(* PLC project prj, KAIST_DSLAB noNameNow 1, author bwkim *)
(* stored: creationDateTime 2018-0-3T10:17:27, modificationDateTime 2018-0-3T10:17:30 *)

PROGRAM program7____wholeTest
  VAR
    FR_PTRIP_TON_copy : null;
  END_VAR
  VAR
    FR_TRIP_TON_copy : null;
  END_VAR
  VAR
    PTRIP_TON : null;
  END_VAR
  VAR
    TRIP_TON : null;
  END_VAR
  VAR
    PTRIP_TON_copy : null;
  END_VAR
  VAR
    TRIP_TON_copy : null;
  END_VAR
  VAR
    PTRIP_TON_copy_copy : null;
  END_VAR
  VAR
    TRIP_TON_copy_copy : null;
  END_VAR
  VAR
    FR_PTRIP_TON_copy_copy : null;
  END_VAR
  VAR
    FR_TRIP_TON_copy_copy : null;
  END_VAR
  VAR
    VF_PTON_copy : null;
  END_VAR
  VAR
    VF_TON_copy : null;
  END_VAR
  VAR
    FR_PTRIP_TON_copy_copy_copy : null;
  END_VAR
  VAR
    FR_TRIP_TON_copy_copy_copy : null;
  END_VAR
  VAR
    FR_PTRIP_TON_copy_copy_copy_copy : null;
  END_VAR
  VAR
    FR_TRIP_TON_copy_copy_copy_copy : null;
  END_VAR
  VAR
    VF_PTON_copy_copy : null;
  END_VAR
  VAR
    VF_TON_copy_copy : null;
  END_VAR
  VAR
    PTRIP_TON_copy_copy_copy : null;
  END_VAR
  VAR
    TRIP_TON_copy_copy_copy : null;
  END_VAR
  VAR
    PTRIP_TON_copy_copy_copy_copy : null;
  END_VAR
  VAR
    TRIP_TON_copy_copy_copy_copy : null;
  END_VAR
  VAR
    FR_PTRIP_TON_copy_copy_copy_copy_copy : null;
  END_VAR
  VAR
    FR_TRIP_TON_copy_copy_copy_copy_copy : null;
  END_VAR
  VAR
    VF_PTON_copy_copy_copy : null;
  END_VAR
  VAR
    VF_TON_copy_copy_copy : null;
  END_VAR
  VAR
    FR_PTRIP_TON_copy_copy_copy_copy_copy_copy : null;
  END_VAR
  VAR
    FR_TRIP_TON_copy_copy_copy_copy_copy_copy : null;
  END_VAR
  VAR_INPUT
    _5_PV_OUT : BOOL := FALSE;
  END_VAR
  VAR_INPUT
    _5_K_DELAY : BOOL := FALSE;
  END_VAR
  VAR_INPUT
    _5_PHYS : BOOL := FALSE;
  END_VAR
  VAR_INPUT
    _5_HYS : BOOL := FALSE;
  END_VAR
  VAR_INPUT
    _5_RNG_MIN : BOOL := FALSE;
  END_VAR
  VAR_INPUT
    _5_RNG_MAX : BOOL := FALSE;
  END_VAR
  VAR_INPUT
    _5_MDL_E : BOOL := FALSE;
  END_VAR
  VAR_INPUT
    _5_AI_E : BOOL := FALSE;
  END_VAR
  VAR_INPUT
    _5_OB_INIT_STA : BOOL := FALSE;
  END_VAR
  VAR_INPUT
    _7_PV_OUT : BOOL := FALSE;
  END_VAR
  VAR_INPUT
    _7_PHYS : BOOL := FALSE;
  END_VAR
  VAR_INPUT
    _7_K_DELAY : BOOL := FALSE;
  END_VAR
  VAR_INPUT
    _7_HYS : BOOL := FALSE;
  END_VAR
  VAR_INPUT
    _7_RNG_MIN : BOOL := FALSE;
  END_VAR
  VAR_INPUT
    _7_RNG_MAX : BOOL := FALSE;
  END_VAR
  VAR_INPUT
    _7_MDL_E : BOOL := FALSE;
  END_VAR
  VAR_INPUT
    _7_AI_E : BOOL := FALSE;
  END_VAR
  VAR_INPUT
    _7_OB_INIT_STA : BOOL := FALSE;
  END_VAR
  VAR_INPUT
    _9_PV_OUT : BOOL := FALSE;
  END_VAR
  VAR_INPUT
    _9_PK_DELAY : BOOL := FALSE;
  END_VAR
  VAR_INPUT
    _9_PHYS : BOOL := FALSE;
  END_VAR
  VAR_INPUT
    _9_K_DELAY : BOOL := FALSE;
  END_VAR
  VAR_INPUT
    _9_HYS : BOOL := FALSE;
  END_VAR
  VAR_INPUT
    _9_RNG_MIN : BOOL := FALSE;
  END_VAR
  VAR_INPUT
    _9_RNG_MAX : BOOL := FALSE;
  END_VAR
  VAR_INPUT
    _9_MDL_E : BOOL := FALSE;
  END_VAR
  VAR_INPUT
    _9_AI_E : BOOL := FALSE;
  END_VAR
  VAR_INPUT
    _9_OB_INIT_STA : BOOL := FALSE;
  END_VAR
  VAR_INPUT
    _B_PV_OUT : BOOL := FALSE;
  END_VAR
  VAR_INPUT
    _B_K_DELAY : BOOL := FALSE;
  END_VAR
  VAR_INPUT
    _B_HYS : BOOL := FALSE;
  END_VAR
  VAR_INPUT
    _B_RNG_MIN : BOOL := FALSE;
  END_VAR
  VAR_INPUT
    _B_RNG_MAX : BOOL := FALSE;
  END_VAR
  VAR_INPUT
    _B_MDL_E : BOOL := FALSE;
  END_VAR
  VAR_INPUT
    _B_AI_E : BOOL := FALSE;
  END_VAR
  VAR_INPUT
    _B_OB_INIT_STA : BOOL := FALSE;
  END_VAR
  VAR_INPUT
    _D_RATE_LMT : BOOL := FALSE;
  END_VAR
  VAR_INPUT
    _D_PV_OUT : BOOL := FALSE;
  END_VAR
  VAR_INPUT
    _D_PV2TSP_DIFF : BOOL := FALSE;
  END_VAR
  VAR_INPUT
    _D_TSP_PRETRIP : BOOL := FALSE;
  END_VAR
  VAR_INPUT
    _D_RATE_TSP_MIN : BOOL := FALSE;
  END_VAR
  VAR_INPUT
    _D_PTSP_PRETRIP : BOOL := FALSE;
  END_VAR
  VAR_INPUT
    _D_TSP2PTSP_DIFF : BOOL := FALSE;
  END_VAR
  VAR_INPUT
    _D_HYS : BOOL := FALSE;
  END_VAR
  VAR_INPUT
    _D_RNG_MIN : BOOL := FALSE;
  END_VAR
  VAR_INPUT
    _D_RNG_MAX : BOOL := FALSE;
  END_VAR
  VAR_INPUT
    _D_MDL_E : BOOL := FALSE;
  END_VAR
  VAR_INPUT
    _D_AI_E : BOOL := FALSE;
  END_VAR
  VAR_INPUT
    _D_OB_INIT_STA : BOOL := FALSE;
  END_VAR
  VAR_INPUT
    _F_PV_OUT : BOOL := FALSE;
  END_VAR
  VAR_INPUT
    _F_K_DELAY : BOOL := FALSE;
  END_VAR
  VAR_INPUT
    _F_HYS : BOOL := FALSE;
  END_VAR
  VAR_INPUT
    _F_RNG_MIN : BOOL := FALSE;
  END_VAR
  VAR_INPUT
    _F_RNG_MAX : BOOL := FALSE;
  END_VAR
  VAR_INPUT
    _F_MDL_E : BOOL := FALSE;
  END_VAR
  VAR_INPUT
    _F_AI_E : BOOL := FALSE;
  END_VAR
  VAR_INPUT
    _F_OB_INIT_STA : BOOL := FALSE;
  END_VAR
  VAR_INPUT
    _G_PV_OUT : BOOL := FALSE;
  END_VAR
  VAR_INPUT
    _G_K_DELAY : BOOL := FALSE;
  END_VAR
  VAR_INPUT
    _G_PHYS : BOOL := FALSE;
  END_VAR
  VAR_INPUT
    _G_HYS : BOOL := FALSE;
  END_VAR
  VAR_INPUT
    _G_RNG_MIN : BOOL := FALSE;
  END_VAR
  VAR_INPUT
    _G_RNG_MAX : BOOL := FALSE;
  END_VAR
  VAR_INPUT
    _G_MDL_E : BOOL := FALSE;
  END_VAR
  VAR_INPUT
    _G_AI_E : BOOL := FALSE;
  END_VAR
  VAR_INPUT
    _G_OB_INIT_STA : BOOL := FALSE;
  END_VAR
  VAR_INPUT
    _6_RATE_LMT : BOOL := FALSE;
  END_VAR
  VAR_INPUT
    _6_PV_OUT : BOOL := FALSE;
  END_VAR
  VAR_INPUT
    _6_PV2TSP_DIFF : BOOL := FALSE;
  END_VAR
  VAR_INPUT
    _6_RATE_TSP_MIN : BOOL := FALSE;
  END_VAR
  VAR_INPUT
    _6_TSP2PTSP_DIFF : BOOL := FALSE;
  END_VAR
  VAR_INPUT
    _6_K_DELAY : BOOL := FALSE;
  END_VAR
  VAR_INPUT
    _6_HYS : BOOL := FALSE;
  END_VAR
  VAR_INPUT
    _6_RNG_MIN : BOOL := FALSE;
  END_VAR
  VAR_INPUT
    _6_RNG_MAX : BOOL := FALSE;
  END_VAR
  VAR_INPUT
    _6_MDL_E : BOOL := FALSE;
  END_VAR
  VAR_INPUT
    _6_AI_E : BOOL := FALSE;
  END_VAR
  VAR_INPUT
    _6_OB_INIT_STA : BOOL := FALSE;
  END_VAR
  VAR_INPUT
    _8_PV_OUT : BOOL := FALSE;
  END_VAR
  VAR_INPUT
    _8_PK_DELAY : BOOL := FALSE;
  END_VAR
  VAR_INPUT
    _8_PHYS : BOOL := FALSE;
  END_VAR
  VAR_INPUT
    _8_K_DELAY : BOOL := FALSE;
  END_VAR
  VAR_INPUT
    _8_HYS : BOOL := FALSE;
  END_VAR
  VAR_INPUT
    _8_RNG_MIN : BOOL := FALSE;
  END_VAR
  VAR_INPUT
    _8_RNG_MAX : BOOL := FALSE;
  END_VAR
  VAR_INPUT
    _8_MDL_E : BOOL := FALSE;
  END_VAR
  VAR_INPUT
    _8_AI_E : BOOL := FALSE;
  END_VAR
  VAR_INPUT
    _8_OB_INIT_STA : BOOL := FALSE;
  END_VAR
  VAR_INPUT
    _A_PV_OUT : BOOL := FALSE;
  END_VAR
  VAR_INPUT
    _A_PK_DELAY : BOOL := FALSE;
  END_VAR
  VAR_INPUT
    _A_PHYS : BOOL := FALSE;
  END_VAR
  VAR_INPUT
    _A_K_DELAY : BOOL := FALSE;
  END_VAR
  VAR_INPUT
    _A_HYS : BOOL := FALSE;
  END_VAR
  VAR_INPUT
    _A_RNG_MIN : BOOL := FALSE;
  END_VAR
  VAR_INPUT
    _A_RNG_MAX : BOOL := FALSE;
  END_VAR
  VAR_INPUT
    _A_MDL_E : BOOL := FALSE;
  END_VAR
  VAR_INPUT
    _A_AI_E : BOOL := FALSE;
  END_VAR
  VAR_INPUT
    _A_OB_INIT_STA : BOOL := FALSE;
  END_VAR
  VAR_INPUT
    _C_PV_OUT : BOOL := FALSE;
  END_VAR
  VAR_INPUT
    _C_K_DELAY : BOOL := FALSE;
  END_VAR
  VAR_INPUT
    _C_PHYS : BOOL := FALSE;
  END_VAR
  VAR_INPUT
    _C_HYS : BOOL := FALSE;
  END_VAR
  VAR_INPUT
    _C_RNG_MIN : BOOL := FALSE;
  END_VAR
  VAR_INPUT
    _C_RNG_MAX : BOOL := FALSE;
  END_VAR
  VAR_INPUT
    _C_MDL_E : BOOL := FALSE;
  END_VAR
  VAR_INPUT
    _C_AI_E : BOOL := FALSE;
  END_VAR
  VAR_INPUT
    _C_OB_INIT_STA : BOOL := FALSE;
  END_VAR
  VAR_INPUT
    _E_RATE_LMT : BOOL := FALSE;
  END_VAR
  VAR_INPUT
    _E_PV_OUT : BOOL := FALSE;
  END_VAR
  VAR_INPUT
    _E_PV2TSP_DIFF : BOOL := FALSE;
  END_VAR
  VAR_INPUT
    _E_TSP_PRETRIP : BOOL := FALSE;
  END_VAR
  VAR_INPUT
    _E_RATE_TSP_MIN : BOOL := FALSE;
  END_VAR
  VAR_INPUT
    _E_PTSP_PRETRIP : BOOL := FALSE;
  END_VAR
  VAR_INPUT
    _E_TSP2PTSP_DIFF : BOOL := FALSE;
  END_VAR
  VAR_INPUT
    _E_K_DELAY : BOOL := FALSE;
  END_VAR
  VAR_INPUT
    _E_HYS : BOOL := FALSE;
  END_VAR
  VAR_INPUT
    _E_RNG_MIN : BOOL := FALSE;
  END_VAR
  VAR_INPUT
    _E_RNG_MAX : BOOL := FALSE;
  END_VAR
  VAR_INPUT
    _E_MDL_E : BOOL := FALSE;
  END_VAR
  VAR_INPUT
    _E_AI_E : BOOL := FALSE;
  END_VAR
  VAR_INPUT
    _E_OB_INIT_STA : BOOL := FALSE;
  END_VAR
  VAR_INPUT
    _2_PV_OUT : BOOL := FALSE;
  END_VAR
  VAR_INPUT
    _2_K_DELAY : BOOL := FALSE;
  END_VAR
  VAR_INPUT
    _2_PHYS : BOOL := FALSE;
  END_VAR
  VAR_INPUT
    _2_HYS : BOOL := FALSE;
  END_VAR
  VAR_INPUT
    _2_RNG_MIN : BOOL := FALSE;
  END_VAR
  VAR_INPUT
    _2_RNG_MAX : BOOL := FALSE;
  END_VAR
  VAR_INPUT
    _2_MDL_E : BOOL := FALSE;
  END_VAR
  VAR_INPUT
    _2_AI_E : BOOL := FALSE;
  END_VAR
  VAR_INPUT
    _2_OB_INIT_STA : BOOL := FALSE;
  END_VAR
  VAR_OUTPUT
    _5_PTON_et : BOOL := FALSE;
  END_VAR
  VAR_OUTPUT
    _5_TON_et : BOOL := FALSE;
  END_VAR
  VAR_OUTPUT
    _7_TON_et : BOOL := FALSE;
  END_VAR
  VAR_OUTPUT
    _9_PTON_et : BOOL := FALSE;
  END_VAR
  VAR_OUTPUT
    _9_TON_et : BOOL := FALSE;
  END_VAR
  VAR_OUTPUT
    _B_PTON_et : BOOL := FALSE;
  END_VAR
  VAR_OUTPUT
    _B_TON_et : BOOL := FALSE;
  END_VAR
  VAR_OUTPUT
    _D_PTON_et : BOOL := FALSE;
  END_VAR
  VAR_OUTPUT
    _D_TON_et : BOOL := FALSE;
  END_VAR
  VAR_OUTPUT
    _F_PTON_et : BOOL := FALSE;
  END_VAR
  VAR_OUTPUT
    _F_TON_et : BOOL := FALSE;
  END_VAR
  VAR_OUTPUT
    _G_PTON_et : BOOL := FALSE;
  END_VAR
  VAR_OUTPUT
    _G_TON_et : BOOL := FALSE;
  END_VAR
  VAR_OUTPUT
    _6_TON_et : BOOL := FALSE;
  END_VAR
  VAR_OUTPUT
    _6_PTON_et : BOOL := FALSE;
  END_VAR
  VAR_OUTPUT
    _8_PTON_et : BOOL := FALSE;
  END_VAR
  VAR_OUTPUT
    _8_TON_et : BOOL := FALSE;
  END_VAR
  VAR_OUTPUT
    _A_PTON_et : BOOL := FALSE;
  END_VAR
  VAR_OUTPUT
    _A_TON_et : BOOL := FALSE;
  END_VAR
  VAR_OUTPUT
    _C_PTON_et : BOOL := FALSE;
  END_VAR
  VAR_OUTPUT
    _C_TON_et : BOOL := FALSE;
  END_VAR
  VAR_OUTPUT
    _E_PTON_et : BOOL := FALSE;
  END_VAR
  VAR_OUTPUT
    _E_TON_et : BOOL := FALSE;
  END_VAR
  VAR_OUTPUT
    _2_PTON_et : BOOL := FALSE;
  END_VAR
  VAR_OUTPUT
    _2_TON_et : BOOL := FALSE;
  END_VAR
  VAR_OUTPUT
    TRIP : BOOL := FALSE;
  END_VAR
  VAR_OUTPUT
    PTRIP : BOOL := FALSE;
  END_VAR
  VAR_IN_OUT
    _5_PTSP : BOOL := FALSE;
  END_VAR
  VAR_IN_OUT
    _5_PTRIP_LOGIC : BOOL := FALSE;
  END_VAR
  VAR_IN_OUT
    _5_TSP : BOOL := FALSE;
  END_VAR
  VAR_IN_OUT
    _5_TRIP_LOGIC : BOOL := FALSE;
  END_VAR
  VAR_IN_OUT
    _7_PTSP : BOOL := FALSE;
  END_VAR
  VAR_IN_OUT
    _7_PTRIP_LOGIC : BOOL := FALSE;
  END_VAR
  VAR_IN_OUT
    _7_PK_DELAY : BOOL := FALSE;
  END_VAR
  VAR_IN_OUT
    _7_PTON_et : BOOL := FALSE;
  END_VAR
  VAR_IN_OUT
    _7_TSP : BOOL := FALSE;
  END_VAR
  VAR_IN_OUT
    _7_TRIP_LOGIC : BOOL := FALSE;
  END_VAR
  VAR_IN_OUT
    _9_PTSP : BOOL := FALSE;
  END_VAR
  VAR_IN_OUT
    _9_PTRIP_LOGIC : BOOL := FALSE;
  END_VAR
  VAR_IN_OUT
    _9_TSP : BOOL := FALSE;
  END_VAR
  VAR_IN_OUT
    _9_TRIP_LOGIC : BOOL := FALSE;
  END_VAR
  VAR_IN_OUT
    _B_PTSP : BOOL := FALSE;
  END_VAR
  VAR_IN_OUT
    _B_PTRIP_LOGIC : BOOL := FALSE;
  END_VAR
  VAR_IN_OUT
    _B_PHYS : BOOL := FALSE;
  END_VAR
  VAR_IN_OUT
    _B_TSP : BOOL := FALSE;
  END_VAR
  VAR_IN_OUT
    _B_TRIP_LOGIC : BOOL := FALSE;
  END_VAR
  VAR_IN_OUT
    _D_TRIP : BOOL := FALSE;
  END_VAR
  VAR_IN_OUT
    _D_PTRIP_LOGIC : BOOL := FALSE;
  END_VAR
  VAR_IN_OUT
    _D_K_DELAY : BOOL := FALSE;
  END_VAR
  VAR_IN_OUT
    _D_TRIP_LOGIC : BOOL := FALSE;
  END_VAR
  VAR_IN_OUT
    _D_TSP : BOOL := FALSE;
  END_VAR
  VAR_IN_OUT
    _D_PTSP : BOOL := FALSE;
  END_VAR
  VAR_IN_OUT
    _F_PTSP : BOOL := FALSE;
  END_VAR
  VAR_IN_OUT
    _F_PTRIP_LOGIC : BOOL := FALSE;
  END_VAR
  VAR_IN_OUT
    _F_PHYS : BOOL := FALSE;
  END_VAR
  VAR_IN_OUT
    _F_TSP : BOOL := FALSE;
  END_VAR
  VAR_IN_OUT
    _F_TRIP_LOGIC : BOOL := FALSE;
  END_VAR
  VAR_IN_OUT
    _G_PTSP : BOOL := FALSE;
  END_VAR
  VAR_IN_OUT
    _G_PTRIP_LOGIC : BOOL := FALSE;
  END_VAR
  VAR_IN_OUT
    _G_TSP : BOOL := FALSE;
  END_VAR
  VAR_IN_OUT
    _G_TRIP_LOGIC : BOOL := FALSE;
  END_VAR
  VAR_IN_OUT
    _6_TSP_PRETRIP : BOOL := FALSE;
  END_VAR
  VAR_IN_OUT
    _6_TRIP : BOOL := FALSE;
  END_VAR
  VAR_IN_OUT
    _6_PTSP_PRETRIP : BOOL := FALSE;
  END_VAR
  VAR_IN_OUT
    _6_PTRIP_LOGIC : BOOL := FALSE;
  END_VAR
  VAR_IN_OUT
    _6_TRIP_LOGIC : BOOL := FALSE;
  END_VAR
  VAR_IN_OUT
    _6_TSP : BOOL := FALSE;
  END_VAR
  VAR_IN_OUT
    _6_PTSP : BOOL := FALSE;
  END_VAR
  VAR_IN_OUT
    _6_PTRIP : BOOL := FALSE;
  END_VAR
  VAR_IN_OUT
    _D_PTRIP : BOOL := FALSE;
  END_VAR
  VAR_IN_OUT
    _8_PTSP : BOOL := FALSE;
  END_VAR
  VAR_IN_OUT
    _8_PTRIP_LOGIC : BOOL := FALSE;
  END_VAR
  VAR_IN_OUT
    _8_TSP : BOOL := FALSE;
  END_VAR
  VAR_IN_OUT
    _8_TRIP_LOGIC : BOOL := FALSE;
  END_VAR
  VAR_IN_OUT
    _A_PTSP : BOOL := FALSE;
  END_VAR
  VAR_IN_OUT
    _A_PTRIP_LOGIC : BOOL := FALSE;
  END_VAR
  VAR_IN_OUT
    _A_TSP : BOOL := FALSE;
  END_VAR
  VAR_IN_OUT
    _A_TRIP_LOGIC : BOOL := FALSE;
  END_VAR
  VAR_IN_OUT
    _C_PTSP : BOOL := FALSE;
  END_VAR
  VAR_IN_OUT
    _C_PTRIP_LOGIC : BOOL := FALSE;
  END_VAR
  VAR_IN_OUT
    _C_TSP : BOOL := FALSE;
  END_VAR
  VAR_IN_OUT
    _C_TRIP_LOGIC : BOOL := FALSE;
  END_VAR
  VAR_IN_OUT
    _E_TRIP : BOOL := FALSE;
  END_VAR
  VAR_IN_OUT
    _E_PTRIP_LOGIC : BOOL := FALSE;
  END_VAR
  VAR_IN_OUT
    _E_TRIP_LOGIC : BOOL := FALSE;
  END_VAR
  VAR_IN_OUT
    _E_TSP : BOOL := FALSE;
  END_VAR
  VAR_IN_OUT
    _E_PTSP : BOOL := FALSE;
  END_VAR
  VAR_IN_OUT
    _2_PTSP : BOOL := FALSE;
  END_VAR
  VAR_IN_OUT
    _2_PTRIP_LOGIC : BOOL := FALSE;
  END_VAR
  VAR_IN_OUT
    _2_TSP : BOOL := FALSE;
  END_VAR
  VAR_IN_OUT
    _2_TRIP_LOGIC : BOOL := FALSE;
  END_VAR
  VAR_IN_OUT
    _E_PTRIP : BOOL := FALSE;
  END_VAR
  VAR  (* added by the conversion: wires and edge detectors of the diagram *)
    _SEL_BOOL660_OUT : BOOL;
    _SEL_BOOL662_OUT : BOOL;
    _SEL_REAL663_OUT : BOOL;
    _AND2_BOOL472_OUT : BOOL;
    _SEL_REAL661_OUT : BOOL;
    _AND2_BOOL474_OUT : BOOL;
    _SEL_BOOL664_OUT : BOOL;
    _SEL_BOOL666_OUT : BOOL;
    _SEL_REAL667_OUT : BOOL;
    _AND2_BOOL478_OUT : BOOL;
    _SEL_REAL665_OUT : BOOL;
    _AND2_BOOL480_OUT : BOOL;
    _SEL_BOOL668_OUT : BOOL;
    _SEL_BOOL670_OUT : BOOL;
    _SEL_REAL671_OUT : BOOL;
    _AND2_BOOL484_OUT : BOOL;
    _SEL_REAL669_OUT : BOOL;
    _AND2_BOOL486_OUT : BOOL;
    _SEL_BOOL672_OUT : BOOL;
    _SEL_BOOL674_OUT : BOOL;
    _SEL_REAL675_OUT : BOOL;
    _AND2_BOOL490_OUT : BOOL;
    _SEL_REAL673_OUT : BOOL;
    _AND2_BOOL492_OUT : BOOL;
    _SUB_REAL612_OUT : BOOL;
    _DIV_REAL772_OUT : BOOL;
    _SEL_REAL864_OUT : BOOL;
    _SEL_REAL865_OUT : BOOL;
    _SEL_REAL866_OUT : BOOL;
    _SEL_BOOL867_OUT : BOOL;
    _SEL_REAL617_OUT : BOOL;
    _SEL_BOOL906_OUT : BOOL;
    _SEL_REAL907_OUT : BOOL;
    _AND2_BOOL810_OUT : BOOL;
    _SEL_REAL910_OUT : BOOL;
    _SEL_REAL911_OUT : BOOL;
    _AND2_BOOL619_OUT : BOOL;
    _AND2_BOOL849_OUT : BOOL;
    _AND2_BOOL850_OUT : BOOL;
    _SEL_BOOL620_OUT : BOOL;
    _SEL_BOOL622_OUT : BOOL;
    _SEL_REAL623_OUT : BOOL;
    _AND2_BOOL450_OUT : BOOL;
    _SEL_REAL621_OUT : BOOL;
    _AND2_BOOL452_OUT : BOOL;
    _SEL_BOOL624_OUT : BOOL;
    _SEL_BOOL626_OUT : BOOL;
    _SEL_REAL627_OUT : BOOL;
    _AND2_BOOL456_OUT : BOOL;
    _SEL_REAL625_OUT : BOOL;
    _AND2_BOOL458_OUT : BOOL;
    _SUB_REAL552_OUT : BOOL;
    _DIV_REAL750_OUT : BOOL;
    _SEL_REAL852_OUT : BOOL;
    _SEL_REAL853_OUT : BOOL;
    _SEL_REAL854_OUT : BOOL;
    _SEL_BOOL855_OUT : BOOL;
    _SEL_REAL557_OUT : BOOL;
    _SEL_BOOL884_OUT : BOOL;
    _SEL_REAL885_OUT : BOOL;
    _AND2_BOOL779_OUT : BOOL;
    _SEL_REAL888_OUT : BOOL;
    _SEL_REAL889_OUT : BOOL;
    _AND2_BOOL559_OUT : BOOL;
    _AND2_BOOL824_OUT : BOOL;
    _AND2_BOOL825_OUT : BOOL;
    _SEL_BOOL560_OUT : BOOL;
    _SEL_BOOL562_OUT : BOOL;
    _SEL_REAL563_OUT : BOOL;
    _AND2_BOOL406_OUT : BOOL;
    _SEL_REAL561_OUT : BOOL;
    _AND2_BOOL408_OUT : BOOL;
    _SEL_BOOL564_OUT : BOOL;
    _SEL_BOOL566_OUT : BOOL;
    _SEL_REAL567_OUT : BOOL;
    _AND2_BOOL412_OUT : BOOL;
    _SEL_REAL565_OUT : BOOL;
    _AND2_BOOL414_OUT : BOOL;
    _SEL_BOOL568_OUT : BOOL;
    _SEL_BOOL570_OUT : BOOL;
    _SEL_REAL571_OUT : BOOL;
    _AND2_BOOL418_OUT : BOOL;
    _SEL_REAL569_OUT : BOOL;
    _AND2_BOOL420_OUT : BOOL;
    _SUB_REAL573_OUT : BOOL;
    _DIV_REAL753_OUT : BOOL;
    _SEL_REAL858_OUT : BOOL;
    _SEL_REAL859_OUT : BOOL;
    _SEL_REAL860_OUT : BOOL;
    _SEL_BOOL861_OUT : BOOL;
    _SEL_REAL578_OUT : BOOL;
    _SEL_BOOL893_OUT : BOOL;
    _SEL_REAL894_OUT : BOOL;
    _AND2_BOOL798_OUT : BOOL;
    _SEL_REAL897_OUT : BOOL;
    _SEL_REAL898_OUT : BOOL;
    _AND2_BOOL580_OUT : BOOL;
    _AND2_BOOL830_OUT : BOOL;
    _AND2_BOOL831_OUT : BOOL;
    _SEL_BOOL581_OUT : BOOL;
    _SEL_BOOL583_OUT : BOOL;
    _SEL_REAL584_OUT : BOOL;
    _AND2_BOOL426_OUT : BOOL;
    _SEL_REAL582_OUT : BOOL;
    _AND2_BOOL428_OUT : BOOL;
    _AND2_BOOL469_OUT : BOOL;
    _AND2_BOOL461_OUT : BOOL;
    _AND2_BOOL463_OUT : BOOL;
    _AND2_BOOL466_OUT : BOOL;
    _AND2_BOOL496_OUT : BOOL;
    _AND2_BOOL499_OUT : BOOL;
    _AND2_BOOL530_OUT : BOOL;
    _AND2_BOOL532_OUT : BOOL;
    _AND2_BOOL534_OUT : BOOL;
    _AND2_BOOL537_OUT : BOOL;
  END_VAR

(* LD diagram, written out as Structured Text *)
FR_PTRIP_TON_copy(IN := AND2_BOOL(GE_REAL(_5_PV_OUT, _5_PTSP), NOT _5_PTRIP_LOGIC), PT := _5_K_DELAY);
_SEL_BOOL660_OUT := SEL_BOOL(FR_PTRIP_TON_copy.Q, _5_PTRIP_LOGIC, TRUE);
_5_PTRIP_LOGIC := _SEL_BOOL660_OUT;
_5_PTON_et := FR_PTRIP_TON_copy.ET;
FR_TRIP_TON_copy(IN := AND2_BOOL(GE_REAL(_5_PV_OUT, _5_TSP), NOT _5_TRIP_LOGIC), PT := _5_K_DELAY);
_SEL_BOOL662_OUT := SEL_BOOL(FR_TRIP_TON_copy.Q, _5_TRIP_LOGIC, TRUE);
_5_TRIP_LOGIC := _SEL_BOOL662_OUT;
_5_TON_et := FR_TRIP_TON_copy.ET;
_SEL_REAL663_OUT := SEL_REAL(FR_TRIP_TON_copy.Q, _5_TSP, SUB_REAL(_5_TSP, _5_HYS));
_AND2_BOOL472_OUT := AND2_BOOL(LT_REAL(_5_PV_OUT, _SEL_REAL663_OUT), _SEL_BOOL662_OUT);
_5_TSP := SEL_REAL(_AND2_BOOL472_OUT, _SEL_REAL663_OUT, ADD2_REAL(_SEL_REAL663_OUT, _5_HYS));
_SEL_REAL661_OUT := SEL_REAL(FR_PTRIP_TON_copy.Q, _5_PTSP, SUB_REAL(_5_PTSP, _5_PHYS));
_AND2_BOOL474_OUT := AND2_BOOL(LT_REAL(_5_PV_OUT, _SEL_REAL661_OUT), _SEL_BOOL660_OUT);
_5_PTSP := SEL_REAL(_AND2_BOOL474_OUT, _SEL_REAL661_OUT, ADD2_REAL(_SEL_REAL661_OUT, _5_PHYS));
PTRIP_TON_copy(IN := AND2_BOOL(LE_REAL(_7_PV_OUT, _7_PTSP), NOT _7_PTRIP_LOGIC), PT := _7_PK_DELAY);
_SEL_BOOL664_OUT := SEL_BOOL(PTRIP_TON_copy.Q, _7_PTRIP_LOGIC, TRUE);
_7_PTRIP_LOGIC := _SEL_BOOL664_OUT;
_7_PTON_et := PTRIP_TON_copy.ET;
TRIP_TON_copy(IN := AND2_BOOL(LE_REAL(_7_PV_OUT, _7_TSP), NOT _7_TRIP_LOGIC), PT := _7_K_DELAY);
_SEL_BOOL666_OUT := SEL_BOOL(TRIP_TON_copy.Q, _7_TRIP_LOGIC, TRUE);
_7_TRIP_LOGIC := _SEL_BOOL666_OUT;
_7_TON_et := TRIP_TON_copy.ET;
_SEL_REAL667_OUT := SEL_REAL(TRIP_TON_copy.Q, _7_TSP, ADD2_REAL(_7_TSP, _7_HYS));
_AND2_BOOL478_OUT := AND2_BOOL(GT_REAL(_7_PV_OUT, _SEL_REAL667_OUT), _SEL_BOOL666_OUT);
_7_TSP := SEL_REAL(_AND2_BOOL478_OUT, _SEL_REAL667_OUT, SUB_REAL(_SEL_REAL667_OUT, _7_HYS));
_SEL_REAL665_OUT := SEL_REAL(PTRIP_TON_copy.Q, _7_PTSP, ADD2_REAL(_7_PTSP, _7_PHYS));
_AND2_BOOL480_OUT := AND2_BOOL(GT_REAL(_7_PV_OUT, _SEL_REAL665_OUT), _SEL_BOOL664_OUT);
_7_PTSP := SEL_REAL(_AND2_BOOL480_OUT, _SEL_REAL665_OUT, SUB_REAL(_SEL_REAL665_OUT, _7_PHYS));
PTRIP_TON_copy_copy(IN := AND2_BOOL(LE_REAL(_9_PV_OUT, _9_PTSP), NOT _9_PTRIP_LOGIC), PT := _9_PK_DELAY);
_SEL_BOOL668_OUT := SEL_BOOL(PTRIP_TON_copy_copy.Q, _9_PTRIP_LOGIC, TRUE);
_9_PTRIP_LOGIC := _SEL_BOOL668_OUT;
_9_PTON_et := PTRIP_TON_copy_copy.ET;
TRIP_TON_copy_copy(IN := AND2_BOOL(LE_REAL(_9_PV_OUT, _9_TSP), NOT _9_TRIP_LOGIC), PT := _9_K_DELAY);
_SEL_BOOL670_OUT := SEL_BOOL(TRIP_TON_copy_copy.Q, _9_TRIP_LOGIC, TRUE);
_9_TRIP_LOGIC := _SEL_BOOL670_OUT;
_9_TON_et := TRIP_TON_copy_copy.ET;
_SEL_REAL671_OUT := SEL_REAL(TRIP_TON_copy_copy.Q, _9_TSP, ADD2_REAL(_9_TSP, _9_HYS));
_AND2_BOOL484_OUT := AND2_BOOL(GT_REAL(_9_PV_OUT, _SEL_REAL671_OUT), _SEL_BOOL670_OUT);
_9_TSP := SEL_REAL(_AND2_BOOL484_OUT, _SEL_REAL671_OUT, SUB_REAL(_SEL_REAL671_OUT, _9_HYS));
_SEL_REAL669_OUT := SEL_REAL(PTRIP_TON_copy_copy.Q, _9_PTSP, ADD2_REAL(_9_PTSP, _9_PHYS));
_AND2_BOOL486_OUT := AND2_BOOL(GT_REAL(_9_PV_OUT, _SEL_REAL669_OUT), _SEL_BOOL668_OUT);
_9_PTSP := SEL_REAL(_AND2_BOOL486_OUT, _SEL_REAL669_OUT, SUB_REAL(_SEL_REAL669_OUT, _9_PHYS));
FR_PTRIP_TON_copy_copy(IN := AND2_BOOL(GE_REAL(_B_PV_OUT, _B_PTSP), NOT _B_PTRIP_LOGIC), PT := _B_K_DELAY);
_SEL_BOOL672_OUT := SEL_BOOL(FR_PTRIP_TON_copy_copy.Q, _B_PTRIP_LOGIC, TRUE);
_B_PTRIP_LOGIC := _SEL_BOOL672_OUT;
_B_PTON_et := FR_PTRIP_TON_copy_copy.ET;
FR_TRIP_TON_copy_copy(IN := AND2_BOOL(GE_REAL(_B_PV_OUT, _B_TSP), NOT _B_TRIP_LOGIC), PT := _B_K_DELAY);
_SEL_BOOL674_OUT := SEL_BOOL(FR_TRIP_TON_copy_copy.Q, _B_TRIP_LOGIC, TRUE);
_B_TRIP_LOGIC := _SEL_BOOL674_OUT;
_B_TON_et := FR_TRIP_TON_copy_copy.ET;
_SEL_REAL675_OUT := SEL_REAL(FR_TRIP_TON_copy_copy.Q, _B_TSP, SUB_REAL(_B_TSP, _B_HYS));
_AND2_BOOL490_OUT := AND2_BOOL(LT_REAL(_B_PV_OUT, _SEL_REAL675_OUT), _SEL_BOOL674_OUT);
_B_TSP := SEL_REAL(_AND2_BOOL490_OUT, _SEL_REAL675_OUT, ADD2_REAL(_SEL_REAL675_OUT, _B_HYS));
_SEL_REAL673_OUT := SEL_REAL(FR_PTRIP_TON_copy_copy.Q, _B_PTSP, SUB_REAL(_B_PTSP, _B_PHYS));
_AND2_BOOL492_OUT := AND2_BOOL(LT_REAL(_B_PV_OUT, _SEL_REAL673_OUT), _SEL_BOOL672_OUT);
_B_PTSP := SEL_REAL(_AND2_BOOL492_OUT, _SEL_REAL673_OUT, ADD2_REAL(_SEL_REAL673_OUT, _B_PHYS));
_SUB_REAL612_OUT := SUB_REAL(_D_PV_OUT, _D_PV2TSP_DIFF);
_DIV_REAL772_OUT := DIV_REAL(MUL2_REAL(_D_RATE_LMT, 1000), 60000);
_SEL_REAL864_OUT := SEL_REAL(AND2_BOOL(GT_REAL(ABS_REAL(SUB_REAL(_D_TSP_PRETRIP, _SUB_REAL612_OUT)), _DIV_REAL772_OUT), GT_REAL(_D_TSP_PRETRIP, _SUB_REAL612_OUT)), _SUB_REAL612_OUT, SUB_REAL(_D_TSP_PRETRIP, _DIV_REAL772_OUT));
_SEL_REAL865_OUT := SEL_REAL(LT_REAL(_SEL_REAL864_OUT, _D_RATE_TSP_MIN), _SEL_REAL864_OUT, _D_RATE_TSP_MIN);
_SEL_REAL866_OUT := SEL_REAL(NOT _D_TRIP, _D_PTSP_PRETRIP, ADD2_REAL(_SEL_REAL865_OUT, _D_TSP2PTSP_DIFF));
VF_PTON_copy(IN := AND2_BOOL(LE_REAL(_D_PV_OUT, _SEL_REAL866_OUT), NOT _D_PTRIP_LOGIC), PT := _D_K_DELAY);
_SEL_BOOL867_OUT := SEL_BOOL(VF_PTON_copy.Q, _D_PTRIP_LOGIC, TRUE);
_D_PTRIP_LOGIC := _SEL_BOOL867_OUT;
_D_PTON_et := VF_PTON_copy.ET;
_SEL_REAL617_OUT := SEL_REAL(NOT _D_TRIP, _D_TSP_PRETRIP, _SEL_REAL865_OUT);
VF_TON_copy(IN := AND2_BOOL(LE_REAL(_D_PV_OUT, _SEL_REAL617_OUT), NOT _D_TRIP_LOGIC), PT := _D_K_DELAY);
_SEL_BOOL906_OUT := SEL_BOOL(VF_TON_copy.Q, _D_TRIP_LOGIC, TRUE);
_D_TRIP_LOGIC := _SEL_BOOL906_OUT;
_D_TON_et := VF_TON_copy.ET;
_SEL_REAL907_OUT := SEL_REAL(VF_TON_copy.Q, _SEL_REAL617_OUT, ADD2_REAL(_SEL_REAL617_OUT, _D_HYS));
_AND2_BOOL810_OUT := AND2_BOOL(_SEL_BOOL906_OUT, GT_REAL(_D_PV_OUT, _SEL_REAL907_OUT));
_SEL_REAL910_OUT := SEL_REAL(_AND2_BOOL810_OUT, _SEL_REAL907_OUT, SUB_REAL(_SEL_REAL907_OUT, _D_HYS));
_D_TSP := _SEL_REAL910_OUT;
_SEL_REAL911_OUT := SEL_REAL(_AND2_BOOL810_OUT, SEL_REAL(VF_TON_copy.Q, _SEL_REAL866_OUT, ADD2_REAL(_SEL_REAL907_OUT, _D_TSP2PTSP_DIFF)), ADD2_REAL(_SEL_REAL910_OUT, _D_TSP2PTSP_DIFF));
_D_PTSP := _SEL_REAL911_OUT;
_AND2_BOOL619_OUT := AND2_BOOL(LT_REAL(_D_RNG_MIN, _D_PV_OUT), LT_REAL(_D_PV_OUT, _D_RNG_MAX));
_AND2_BOOL849_OUT := AND2_BOOL(OR4_BOOL(NOT _AND2_BOOL619_OUT, _D_MDL_E, _D_AI_E, SEL_BOOL(AND2_BOOL(_SEL_BOOL867_OUT, GT_REAL(_D_PV_OUT, _SEL_REAL911_OUT)), _SEL_BOOL867_OUT, FALSE)), NOT _D_OB_INIT_STA);
_D_PTRIP := _AND2_BOOL849_OUT;
_AND2_BOOL850_OUT := AND2_BOOL(OR4_BOOL(NOT _AND2_BOOL619_OUT, _D_MDL_E, _D_AI_E, SEL_BOOL(_AND2_BOOL810_OUT, _SEL_BOOL906_OUT, FALSE)), NOT _D_OB_INIT_STA);
_D_TRIP := _AND2_BOOL850_OUT;
FR_PTRIP_TON_copy_copy_copy(IN := AND2_BOOL(GE_REAL(_F_PV_OUT, _F_PTSP), NOT _F_PTRIP_LOGIC), PT := _F_K_DELAY);
_SEL_BOOL620_OUT := SEL_BOOL(FR_PTRIP_TON_copy_copy_copy.Q, _F_PTRIP_LOGIC, TRUE);
_F_PTRIP_LOGIC := _SEL_BOOL620_OUT;
_F_PTON_et := FR_PTRIP_TON_copy_copy_copy.ET;
FR_TRIP_TON_copy_copy_copy(IN := AND2_BOOL(GE_REAL(_F_PV_OUT, _F_TSP), NOT _F_TRIP_LOGIC), PT := _F_K_DELAY);
_SEL_BOOL622_OUT := SEL_BOOL(FR_TRIP_TON_copy_copy_copy.Q, _F_TRIP_LOGIC, TRUE);
_F_TRIP_LOGIC := _SEL_BOOL622_OUT;
_F_TON_et := FR_TRIP_TON_copy_copy_copy.ET;
_SEL_REAL623_OUT := SEL_REAL(FR_TRIP_TON_copy_copy_copy.Q, _F_TSP, SUB_REAL(_F_TSP, _F_HYS));
_AND2_BOOL450_OUT := AND2_BOOL(LT_REAL(_F_PV_OUT, _SEL_REAL623_OUT), _SEL_BOOL622_OUT);
_F_TSP := SEL_REAL(_AND2_BOOL450_OUT, _SEL_REAL623_OUT, ADD2_REAL(_SEL_REAL623_OUT, _F_HYS));
_SEL_REAL621_OUT := SEL_REAL(FR_PTRIP_TON_copy_copy_copy.Q, _F_PTSP, SUB_REAL(_F_PTSP, _F_PHYS));
_AND2_BOOL452_OUT := AND2_BOOL(LT_REAL(_F_PV_OUT, _SEL_REAL621_OUT), _SEL_BOOL620_OUT);
_F_PTSP := SEL_REAL(_AND2_BOOL452_OUT, _SEL_REAL621_OUT, ADD2_REAL(_SEL_REAL621_OUT, _F_PHYS));
FR_PTRIP_TON_copy_copy_copy_copy(IN := AND2_BOOL(GE_REAL(_G_PV_OUT, _G_PTSP), NOT _G_PTRIP_LOGIC), PT := _G_K_DELAY);
_SEL_BOOL624_OUT := SEL_BOOL(FR_PTRIP_TON_copy_copy_copy_copy.Q, _G_PTRIP_LOGIC, TRUE);
_G_PTRIP_LOGIC := _SEL_BOOL624_OUT;
_G_PTON_et := FR_PTRIP_TON_copy_copy_copy_copy.ET;
FR_TRIP_TON_copy_copy_copy_copy(IN := AND2_BOOL(GE_REAL(_G_PV_OUT, _G_TSP), NOT _G_TRIP_LOGIC), PT := _G_K_DELAY);
_SEL_BOOL626_OUT := SEL_BOOL(FR_TRIP_TON_copy_copy_copy_copy.Q, _G_TRIP_LOGIC, TRUE);
_G_TRIP_LOGIC := _SEL_BOOL626_OUT;
_G_TON_et := FR_TRIP_TON_copy_copy_copy_copy.ET;
_SEL_REAL627_OUT := SEL_REAL(FR_TRIP_TON_copy_copy_copy_copy.Q, _G_TSP, SUB_REAL(_G_TSP, _G_HYS));
_AND2_BOOL456_OUT := AND2_BOOL(LT_REAL(_G_PV_OUT, _SEL_REAL627_OUT), _SEL_BOOL626_OUT);
_G_TSP := SEL_REAL(_AND2_BOOL456_OUT, _SEL_REAL627_OUT, ADD2_REAL(_SEL_REAL627_OUT, _G_HYS));
_SEL_REAL625_OUT := SEL_REAL(FR_PTRIP_TON_copy_copy_copy_copy.Q, _G_PTSP, SUB_REAL(_G_PTSP, _G_PHYS));
_AND2_BOOL458_OUT := AND2_BOOL(LT_REAL(_G_PV_OUT, _SEL_REAL625_OUT), _SEL_BOOL624_OUT);
_G_PTSP := SEL_REAL(_AND2_BOOL458_OUT, _SEL_REAL625_OUT, ADD2_REAL(_SEL_REAL625_OUT, _G_PHYS));
_SUB_REAL552_OUT := SUB_REAL(_6_PV_OUT, _6_PV2TSP_DIFF);
_DIV_REAL750_OUT := DIV_REAL(MUL2_REAL(_6_RATE_LMT, 1000), 60000);
_SEL_REAL852_OUT := SEL_REAL(AND2_BOOL(GT_REAL(ABS_REAL(SUB_REAL(_6_TSP_PRETRIP, _SUB_REAL552_OUT)), _DIV_REAL750_OUT), GT_REAL(_6_TSP_PRETRIP, _SUB_REAL552_OUT)), _SUB_REAL552_OUT, SUB_REAL(_6_TSP_PRETRIP, _DIV_REAL750_OUT));
_SEL_REAL853_OUT := SEL_REAL(LT_REAL(_SEL_REAL852_OUT, _6_RATE_TSP_MIN), _SEL_REAL852_OUT, _6_RATE_TSP_MIN);
_SEL_REAL854_OUT := SEL_REAL(NOT _6_TRIP, _6_PTSP_PRETRIP, ADD2_REAL(_SEL_REAL853_OUT, _6_TSP2PTSP_DIFF));
VF_PTON_copy_copy(IN := AND2_BOOL(LE_REAL(_6_PV_OUT, _SEL_REAL854_OUT), NOT _6_PTRIP_LOGIC), PT := _6_K_DELAY);
_SEL_BOOL855_OUT := SEL_BOOL(VF_PTON_copy_copy.Q, _6_PTRIP_LOGIC, TRUE);
_6_PTRIP_LOGIC := _SEL_BOOL855_OUT;
_6_PTON_et := VF_PTON_copy_copy.ET;
_SEL_REAL557_OUT := SEL_REAL(NOT _6_TRIP, _6_TSP_PRETRIP, _SEL_REAL853_OUT);
VF_TON_copy_copy(IN := AND2_BOOL(LE_REAL(_6_PV_OUT, _SEL_REAL557_OUT), NOT _6_TRIP_LOGIC), PT := _6_K_DELAY);
_SEL_BOOL884_OUT := SEL_BOOL(VF_TON_copy_copy.Q, _6_TRIP_LOGIC, TRUE);
_6_TRIP_LOGIC := _SEL_BOOL884_OUT;
_6_TON_et := VF_TON_copy_copy.ET;
_SEL_REAL885_OUT := SEL_REAL(VF_TON_copy_copy.Q, _SEL_REAL557_OUT, ADD2_REAL(_SEL_REAL557_OUT, _6_HYS));
_AND2_BOOL779_OUT := AND2_BOOL(_SEL_BOOL884_OUT, GT_REAL(_6_PV_OUT, _SEL_REAL885_OUT));
_SEL_REAL888_OUT := SEL_REAL(_AND2_BOOL779_OUT, _SEL_REAL885_OUT, SUB_REAL(_SEL_REAL885_OUT, _6_HYS));
_6_TSP := _SEL_REAL888_OUT;
_SEL_REAL889_OUT := SEL_REAL(_AND2_BOOL779_OUT, SEL_REAL(VF_TON_copy_copy.Q, _SEL_REAL854_OUT, ADD2_REAL(_SEL_REAL885_OUT, _6_TSP2PTSP_DIFF)), ADD2_REAL(_SEL_REAL888_OUT, _6_TSP2PTSP_DIFF));
_6_PTSP := _SEL_REAL889_OUT;
_AND2_BOOL559_OUT := AND2_BOOL(LT_REAL(_6_RNG_MIN, _6_PV_OUT), LT_REAL(_6_PV_OUT, _6_RNG_MAX));
_AND2_BOOL824_OUT := AND2_BOOL(OR4_BOOL(NOT _AND2_BOOL559_OUT, _6_MDL_E, _6_AI_E, SEL_BOOL(AND2_BOOL(_SEL_BOOL855_OUT, GT_REAL(_6_PV_OUT, _SEL_REAL889_OUT)), _SEL_BOOL855_OUT, FALSE)), NOT _6_OB_INIT_STA);
_6_PTRIP := _AND2_BOOL824_OUT;
_AND2_BOOL825_OUT := AND2_BOOL(OR4_BOOL(NOT _AND2_BOOL559_OUT, _6_MDL_E, _6_AI_E, SEL_BOOL(_AND2_BOOL779_OUT, _SEL_BOOL884_OUT, FALSE)), NOT _6_OB_INIT_STA);
_6_TRIP := _AND2_BOOL825_OUT;
PTRIP_TON_copy_copy_copy(IN := AND2_BOOL(LE_REAL(_8_PV_OUT, _8_PTSP), NOT _8_PTRIP_LOGIC), PT := _8_PK_DELAY);
_SEL_BOOL560_OUT := SEL_BOOL(PTRIP_TON_copy_copy_copy.Q, _8_PTRIP_LOGIC, TRUE);
_8_PTRIP_LOGIC := _SEL_BOOL560_OUT;
_8_PTON_et := PTRIP_TON_copy_copy_copy.ET;
TRIP_TON_copy_copy_copy(IN := AND2_BOOL(LE_REAL(_8_PV_OUT, _8_TSP), NOT _8_TRIP_LOGIC), PT := _8_K_DELAY);
_SEL_BOOL562_OUT := SEL_BOOL(TRIP_TON_copy_copy_copy.Q, _8_TRIP_LOGIC, TRUE);
_8_TRIP_LOGIC := _SEL_BOOL562_OUT;
_8_TON_et := TRIP_TON_copy_copy_copy.ET;
_SEL_REAL563_OUT := SEL_REAL(TRIP_TON_copy_copy_copy.Q, _8_TSP, ADD2_REAL(_8_TSP, _8_HYS));
_AND2_BOOL406_OUT := AND2_BOOL(GT_REAL(_8_PV_OUT, _SEL_REAL563_OUT), _SEL_BOOL562_OUT);
_8_TSP := SEL_REAL(_AND2_BOOL406_OUT, _SEL_REAL563_OUT, SUB_REAL(_SEL_REAL563_OUT, _8_HYS));
_SEL_REAL561_OUT := SEL_REAL(PTRIP_TON_copy_copy_copy.Q, _8_PTSP, ADD2_REAL(_8_PTSP, _8_PHYS));
_AND2_BOOL408_OUT := AND2_BOOL(GT_REAL(_8_PV_OUT, _SEL_REAL561_OUT), _SEL_BOOL560_OUT);
_8_PTSP := SEL_REAL(_AND2_BOOL408_OUT, _SEL_REAL561_OUT, SUB_REAL(_SEL_REAL561_OUT, _8_PHYS));
PTRIP_TON_copy_copy_copy_copy(IN := AND2_BOOL(LE_REAL(_A_PV_OUT, _A_PTSP), NOT _A_PTRIP_LOGIC), PT := _A_PK_DELAY);
_SEL_BOOL564_OUT := SEL_BOOL(PTRIP_TON_copy_copy_copy_copy.Q, _A_PTRIP_LOGIC, TRUE);
_A_PTRIP_LOGIC := _SEL_BOOL564_OUT;
_A_PTON_et := PTRIP_TON_copy_copy_copy_copy.ET;
TRIP_TON_copy_copy_copy_copy(IN := AND2_BOOL(LE_REAL(_A_PV_OUT, _A_TSP), NOT _A_TRIP_LOGIC), PT := _A_K_DELAY);
_SEL_BOOL566_OUT := SEL_BOOL(TRIP_TON_copy_copy_copy_copy.Q, _A_TRIP_LOGIC, TRUE);
_A_TRIP_LOGIC := _SEL_BOOL566_OUT;
_A_TON_et := TRIP_TON_copy_copy_copy_copy.ET;
_SEL_REAL567_OUT := SEL_REAL(TRIP_TON_copy_copy_copy_copy.Q, _A_TSP, ADD2_REAL(_A_TSP, _A_HYS));
_AND2_BOOL412_OUT := AND2_BOOL(GT_REAL(_A_PV_OUT, _SEL_REAL567_OUT), _SEL_BOOL566_OUT);
_A_TSP := SEL_REAL(_AND2_BOOL412_OUT, _SEL_REAL567_OUT, SUB_REAL(_SEL_REAL567_OUT, _A_HYS));
_SEL_REAL565_OUT := SEL_REAL(PTRIP_TON_copy_copy_copy_copy.Q, _A_PTSP, ADD2_REAL(_A_PTSP, _A_PHYS));
_AND2_BOOL414_OUT := AND2_BOOL(GT_REAL(_A_PV_OUT, _SEL_REAL565_OUT), _SEL_BOOL564_OUT);
_A_PTSP := SEL_REAL(_AND2_BOOL414_OUT, _SEL_REAL565_OUT, SUB_REAL(_SEL_REAL565_OUT, _A_PHYS));
FR_PTRIP_TON_copy_copy_copy_copy_copy(IN := AND2_BOOL(GE_REAL(_C_PV_OUT, _C_PTSP), NOT _C_PTRIP_LOGIC), PT := _C_K_DELAY);
_SEL_BOOL568_OUT := SEL_BOOL(FR_PTRIP_TON_copy_copy_copy_copy_copy.Q, _C_PTRIP_LOGIC, TRUE);
_C_PTRIP_LOGIC := _SEL_BOOL568_OUT;
_C_PTON_et := FR_PTRIP_TON_copy_copy_copy_copy_copy.ET;
FR_TRIP_TON_copy_copy_copy_copy_copy(IN := AND2_BOOL(GE_REAL(_C_PV_OUT, _C_TSP), NOT _C_TRIP_LOGIC), PT := _C_K_DELAY);
_SEL_BOOL570_OUT := SEL_BOOL(FR_TRIP_TON_copy_copy_copy_copy_copy.Q, _C_TRIP_LOGIC, TRUE);
_C_TRIP_LOGIC := _SEL_BOOL570_OUT;
_C_TON_et := FR_TRIP_TON_copy_copy_copy_copy_copy.ET;
_SEL_REAL571_OUT := SEL_REAL(FR_TRIP_TON_copy_copy_copy_copy_copy.Q, _C_TSP, SUB_REAL(_C_TSP, _C_HYS));
_AND2_BOOL418_OUT := AND2_BOOL(LT_REAL(_C_PV_OUT, _SEL_REAL571_OUT), _SEL_BOOL570_OUT);
_C_TSP := SEL_REAL(_AND2_BOOL418_OUT, _SEL_REAL571_OUT, ADD2_REAL(_SEL_REAL571_OUT, _C_HYS));
_SEL_REAL569_OUT := SEL_REAL(FR_PTRIP_TON_copy_copy_copy_copy_copy.Q, _C_PTSP, SUB_REAL(_C_PTSP, _C_PHYS));
_AND2_BOOL420_OUT := AND2_BOOL(LT_REAL(_C_PV_OUT, _SEL_REAL569_OUT), _SEL_BOOL568_OUT);
_C_PTSP := SEL_REAL(_AND2_BOOL420_OUT, _SEL_REAL569_OUT, ADD2_REAL(_SEL_REAL569_OUT, _C_PHYS));
_SUB_REAL573_OUT := SUB_REAL(_E_PV_OUT, _E_PV2TSP_DIFF);
_DIV_REAL753_OUT := DIV_REAL(MUL2_REAL(_E_RATE_LMT, 1000), 60000);
_SEL_REAL858_OUT := SEL_REAL(AND2_BOOL(GT_REAL(ABS_REAL(SUB_REAL(_E_TSP_PRETRIP, _SUB_REAL573_OUT)), _DIV_REAL753_OUT), GT_REAL(_E_TSP_PRETRIP, _SUB_REAL573_OUT)), _SUB_REAL573_OUT, SUB_REAL(_E_TSP_PRETRIP, _DIV_REAL753_OUT));
_SEL_REAL859_OUT := SEL_REAL(LT_REAL(_SEL_REAL858_OUT, _E_RATE_TSP_MIN), _SEL_REAL858_OUT, _E_RATE_TSP_MIN);
_SEL_REAL860_OUT := SEL_REAL(NOT _E_TRIP, _E_PTSP_PRETRIP, ADD2_REAL(_SEL_REAL859_OUT, _E_TSP2PTSP_DIFF));
VF_PTON_copy_copy_copy(IN := AND2_BOOL(LE_REAL(_E_PV_OUT, _SEL_REAL860_OUT), NOT _E_PTRIP_LOGIC), PT := _E_K_DELAY);
_SEL_BOOL861_OUT := SEL_BOOL(VF_PTON_copy_copy_copy.Q, _E_PTRIP_LOGIC, TRUE);
_E_PTRIP_LOGIC := _SEL_BOOL861_OUT;
_E_PTON_et := VF_PTON_copy_copy_copy.ET;
_SEL_REAL578_OUT := SEL_REAL(NOT _E_TRIP, _E_TSP_PRETRIP, _SEL_REAL859_OUT);
VF_TON_copy_copy_copy(IN := AND2_BOOL(LE_REAL(_E_PV_OUT, _SEL_REAL578_OUT), NOT _E_TRIP_LOGIC), PT := _E_K_DELAY);
_SEL_BOOL893_OUT := SEL_BOOL(VF_TON_copy_copy_copy.Q, _E_TRIP_LOGIC, TRUE);
_E_TRIP_LOGIC := _SEL_BOOL893_OUT;
_E_TON_et := VF_TON_copy_copy_copy.ET;
_SEL_REAL894_OUT := SEL_REAL(VF_TON_copy_copy_copy.Q, _SEL_REAL578_OUT, ADD2_REAL(_SEL_REAL578_OUT, _E_HYS));
_AND2_BOOL798_OUT := AND2_BOOL(_SEL_BOOL893_OUT, GT_REAL(_E_PV_OUT, _SEL_REAL894_OUT));
_SEL_REAL897_OUT := SEL_REAL(_AND2_BOOL798_OUT, _SEL_REAL894_OUT, SUB_REAL(_SEL_REAL894_OUT, _E_HYS));
_E_TSP := _SEL_REAL897_OUT;
_SEL_REAL898_OUT := SEL_REAL(_AND2_BOOL798_OUT, SEL_REAL(VF_TON_copy_copy_copy.Q, _SEL_REAL860_OUT, ADD2_REAL(_SEL_REAL894_OUT, _E_TSP2PTSP_DIFF)), ADD2_REAL(_SEL_REAL897_OUT, _E_TSP2PTSP_DIFF));
_E_PTSP := _SEL_REAL898_OUT;
_AND2_BOOL580_OUT := AND2_BOOL(LT_REAL(_E_RNG_MIN, _E_PV_OUT), LT_REAL(_E_PV_OUT, _E_RNG_MAX));
_AND2_BOOL830_OUT := AND2_BOOL(OR4_BOOL(NOT _AND2_BOOL580_OUT, _E_MDL_E, _E_AI_E, SEL_BOOL(AND2_BOOL(_SEL_BOOL861_OUT, GT_REAL(_E_PV_OUT, _SEL_REAL898_OUT)), _SEL_BOOL861_OUT, FALSE)), NOT _E_OB_INIT_STA);
_E_PTRIP := _AND2_BOOL830_OUT;
_AND2_BOOL831_OUT := AND2_BOOL(OR4_BOOL(NOT _AND2_BOOL580_OUT, _E_MDL_E, _E_AI_E, SEL_BOOL(_AND2_BOOL798_OUT, _SEL_BOOL893_OUT, FALSE)), NOT _E_OB_INIT_STA);
_E_TRIP := _AND2_BOOL831_OUT;
FR_PTRIP_TON_copy_copy_copy_copy_copy_copy(IN := AND2_BOOL(GE_REAL(_2_PV_OUT, _2_PTSP), NOT _2_PTRIP_LOGIC), PT := _2_K_DELAY);
_SEL_BOOL581_OUT := SEL_BOOL(FR_PTRIP_TON_copy_copy_copy_copy_copy_copy.Q, _2_PTRIP_LOGIC, TRUE);
_2_PTRIP_LOGIC := _SEL_BOOL581_OUT;
_2_PTON_et := FR_PTRIP_TON_copy_copy_copy_copy_copy_copy.ET;
FR_TRIP_TON_copy_copy_copy_copy_copy_copy(IN := AND2_BOOL(GE_REAL(_2_PV_OUT, _2_TSP), NOT _2_TRIP_LOGIC), PT := _2_K_DELAY);
_SEL_BOOL583_OUT := SEL_BOOL(FR_TRIP_TON_copy_copy_copy_copy_copy_copy.Q, _2_TRIP_LOGIC, TRUE);
_2_TRIP_LOGIC := _SEL_BOOL583_OUT;
_2_TON_et := FR_TRIP_TON_copy_copy_copy_copy_copy_copy.ET;
_SEL_REAL584_OUT := SEL_REAL(FR_TRIP_TON_copy_copy_copy_copy_copy_copy.Q, _2_TSP, SUB_REAL(_2_TSP, _2_HYS));
_AND2_BOOL426_OUT := AND2_BOOL(LT_REAL(_2_PV_OUT, _SEL_REAL584_OUT), _SEL_BOOL583_OUT);
_2_TSP := SEL_REAL(_AND2_BOOL426_OUT, _SEL_REAL584_OUT, ADD2_REAL(_SEL_REAL584_OUT, _2_HYS));
_SEL_REAL582_OUT := SEL_REAL(FR_PTRIP_TON_copy_copy_copy_copy_copy_copy.Q, _2_PTSP, SUB_REAL(_2_PTSP, _2_PHYS));
_AND2_BOOL428_OUT := AND2_BOOL(LT_REAL(_2_PV_OUT, _SEL_REAL582_OUT), _SEL_BOOL581_OUT);
_2_PTSP := SEL_REAL(_AND2_BOOL428_OUT, _SEL_REAL582_OUT, ADD2_REAL(_SEL_REAL582_OUT, _2_PHYS));
_AND2_BOOL469_OUT := AND2_BOOL(LT_REAL(_2_RNG_MIN, _2_PV_OUT), LT_REAL(_2_PV_OUT, _2_RNG_MAX));
_AND2_BOOL461_OUT := AND2_BOOL(LT_REAL(_8_RNG_MIN, _8_PV_OUT), LT_REAL(_8_PV_OUT, _8_RNG_MAX));
_AND2_BOOL463_OUT := AND2_BOOL(LT_REAL(_A_RNG_MIN, _A_PV_OUT), LT_REAL(_A_PV_OUT, _A_RNG_MAX));
_AND2_BOOL466_OUT := AND2_BOOL(LT_REAL(_C_RNG_MIN, _C_PV_OUT), LT_REAL(_C_PV_OUT, _C_RNG_MAX));
_AND2_BOOL496_OUT := AND2_BOOL(LT_REAL(_F_RNG_MIN, _F_PV_OUT), LT_REAL(_F_PV_OUT, _F_RNG_MAX));
_AND2_BOOL499_OUT := AND2_BOOL(LT_REAL(_G_RNG_MIN, _G_PV_OUT), LT_REAL(_G_PV_OUT, _G_RNG_MAX));
_AND2_BOOL530_OUT := AND2_BOOL(LT_REAL(_5_RNG_MIN, _5_PV_OUT), LT_REAL(_5_PV_OUT, _5_RNG_MAX));
_AND2_BOOL532_OUT := AND2_BOOL(LT_REAL(_7_RNG_MIN, _7_PV_OUT), LT_REAL(_7_PV_OUT, _7_RNG_MAX));
_AND2_BOOL534_OUT := AND2_BOOL(LT_REAL(_9_RNG_MIN, _9_PV_OUT), LT_REAL(_9_PV_OUT, _9_RNG_MAX));
_AND2_BOOL537_OUT := AND2_BOOL(LT_REAL(_B_RNG_MIN, _B_PV_OUT), LT_REAL(_B_PV_OUT, _B_RNG_MAX));
PTRIP := OR4_BOOL(OR2_BOOL(_AND2_BOOL830_OUT, AND2_BOOL(OR4_BOOL(_AND2_BOOL469_OUT, _2_MDL_E, _2_AI_E, SEL_BOOL(_AND2_BOOL428_OUT, _SEL_BOOL581_OUT, FALSE)), NOT _2_OB_INIT_STA)), OR3_BOOL(AND2_BOOL(OR4_BOOL(_AND2_BOOL461_OUT, _8_MDL_E, _8_AI_E, SEL_BOOL(_AND2_BOOL408_OUT, _SEL_BOOL560_OUT, FALSE)), NOT _8_OB_INIT_STA), AND2_BOOL(OR4_BOOL(_AND2_BOOL463_OUT, _A_MDL_E, _A_AI_E, SEL_BOOL(_AND2_BOOL414_OUT, _SEL_BOOL564_OUT, FALSE)), NOT _A_OB_INIT_STA), AND2_BOOL(OR4_BOOL(_AND2_BOOL466_OUT, _C_MDL_E, _C_AI_E, SEL_BOOL(_AND2_BOOL420_OUT, _SEL_BOOL568_OUT, FALSE)), NOT _C_OB_INIT_STA)), OR4_BOOL(_AND2_BOOL849_OUT, AND2_BOOL(OR4_BOOL(_AND2_BOOL496_OUT, _F_MDL_E, _F_AI_E, SEL_BOOL(_AND2_BOOL452_OUT, _SEL_BOOL620_OUT, FALSE)), NOT _F_OB_INIT_STA), AND2_BOOL(OR4_BOOL(_AND2_BOOL499_OUT, _G_MDL_E, _G_AI_E, SEL_BOOL(_AND2_BOOL458_OUT, _SEL_BOOL624_OUT, FALSE)), NOT _G_OB_INIT_STA), _AND2_BOOL824_OUT), OR4_BOOL(AND2_BOOL(OR4_BOOL(_AND2_BOOL530_OUT, _5_MDL_E, _5_AI_E, SEL_BOOL(_AND2_BOOL474_OUT, _SEL_BOOL660_OUT, FALSE)), NOT _5_OB_INIT_STA), AND2_BOOL(OR4_BOOL(_AND2_BOOL532_OUT, _7_MDL_E, _7_AI_E, SEL_BOOL(_AND2_BOOL480_OUT, _SEL_BOOL664_OUT, FALSE)), NOT _7_OB_INIT_STA), AND2_BOOL(OR4_BOOL(_AND2_BOOL534_OUT, _9_MDL_E, _9_AI_E, SEL_BOOL(_AND2_BOOL486_OUT, _SEL_BOOL668_OUT, FALSE)), NOT _9_OB_INIT_STA), AND2_BOOL(OR4_BOOL(_AND2_BOOL537_OUT, _B_MDL_E, _B_AI_E, SEL_BOOL(_AND2_BOOL492_OUT, _SEL_BOOL672_OUT, FALSE)), NOT _B_OB_INIT_STA)));
TRIP := OR4_BOOL(OR4_BOOL(AND2_BOOL(OR4_BOOL(_AND2_BOOL530_OUT, _5_MDL_E, _5_AI_E, SEL_BOOL(_AND2_BOOL472_OUT, _SEL_BOOL662_OUT, FALSE)), NOT _5_OB_INIT_STA), AND2_BOOL(OR4_BOOL(_AND2_BOOL532_OUT, _7_MDL_E, _7_AI_E, SEL_BOOL(_AND2_BOOL478_OUT, _SEL_BOOL666_OUT, FALSE)), NOT _7_OB_INIT_STA), AND2_BOOL(OR4_BOOL(_AND2_BOOL534_OUT, _9_MDL_E, _9_AI_E, SEL_BOOL(_AND2_BOOL484_OUT, _SEL_BOOL670_OUT, FALSE)), NOT _9_OB_INIT_STA), AND2_BOOL(OR4_BOOL(_AND2_BOOL537_OUT, _B_MDL_E, _B_AI_E, SEL_BOOL(_AND2_BOOL490_OUT, _SEL_BOOL674_OUT, FALSE)), NOT _B_OB_INIT_STA)), OR4_BOOL(_AND2_BOOL850_OUT, AND2_BOOL(OR4_BOOL(_AND2_BOOL496_OUT, _F_MDL_E, _F_AI_E, SEL_BOOL(_AND2_BOOL450_OUT, _SEL_BOOL622_OUT, FALSE)), NOT _F_OB_INIT_STA), AND2_BOOL(OR4_BOOL(_AND2_BOOL499_OUT, _G_MDL_E, _G_AI_E, SEL_BOOL(_AND2_BOOL456_OUT, _SEL_BOOL626_OUT, FALSE)), NOT _G_OB_INIT_STA), _AND2_BOOL825_OUT), OR3_BOOL(AND2_BOOL(OR4_BOOL(_AND2_BOOL461_OUT, _8_MDL_E, _8_AI_E, SEL_BOOL(_AND2_BOOL406_OUT, _SEL_BOOL562_OUT, FALSE)), NOT _8_OB_INIT_STA), AND2_BOOL(OR4_BOOL(_AND2_BOOL463_OUT, _A_MDL_E, _A_AI_E, SEL_BOOL(_AND2_BOOL412_OUT, _SEL_BOOL566_OUT, FALSE)), NOT _A_OB_INIT_STA), AND2_BOOL(OR4_BOOL(_AND2_BOOL466_OUT, _C_MDL_E, _C_AI_E, SEL_BOOL(_AND2_BOOL418_OUT, _SEL_BOOL570_OUT, FALSE)), NOT _C_OB_INIT_STA)), OR2_BOOL(_AND2_BOOL831_OUT, AND2_BOOL(OR4_BOOL(_AND2_BOOL469_OUT, _2_MDL_E, _2_AI_E, SEL_BOOL(_AND2_BOOL426_OUT, _SEL_BOOL583_OUT, FALSE)), NOT _2_OB_INIT_STA)));
END_PROGRAM
